(* PLC project Generated.project, CODESYS CODESYS V3.5 SP19 Patch 1 *)
(* stored: creationDateTime 2026-09-14T14:47:22.341572, modificationDateTime 2026-09-14T14:47:22.341572 *)

(* ═══════════════════════════════════════════════════════════════ ⚙️ ST_CycleMachineHomingCfg — Réglages IHM du cycle de référencement machine ─────────────────────────────────────────────────────────────── 🎯 Mise en service. Les réglages géométriques (positions capteur, offsets benne) restent portés par GVL_PERSISTENT (_WinchM1CfgPersist / _BucketCfgPersist). 💾 Ponté vers persist (_CycleMachineHomingCfgPersist) via FB_CfgPersistBridge_CycleMachineHomingCfg. ═══════════════════════════════════════════════════════════════ *)
TYPE ST_CycleMachineHomingCfg : STRUCT
  ForceStepTarget : INT := 0;  (* 🔧 Step GRAFCET cible du forçage (0=HX0 .. 9=HXF), borné côté FB *)
  Initialized : BOOL := FALSE;  (* 🚦 flag restauration boot *)
END_STRUCT;
END_TYPE

(* ======================================================================= 💾 FB_CfgPersistBridge_CycleMachineHomingCfg — Pont persistance pour ST_CycleMachineHomingCfg ─────────────────────────────────────────────────────────────── 🎯 Rôle : Restauration et synchronisation bidirectionnelle IHM / Persist 💾 Persistance : Transfert GVL_PERSISTENT <-> GVL_IHM sur Initialized 📄 Doc métier : DOC/AF/AF_Partie-03_Contrats_Composants_v2.3.md §3 ======================================================================= *)
FUNCTION_BLOCK FB_CfgPersistBridge_CycleMachineHomingCfg
  VAR_OUTPUT
    JustRestored : BOOL;  (* === ETATS RESTAURATION === <-- [STAT] Vrai sur le cycle de restauration initiale *)
  END_VAR
  VAR_IN_OUT
    Hmi : ST_CycleMachineHomingCfg;  (* === BUS CONFIGURATION ET PERSISTANCE === <-> [BUS] Structure de configuration IHM *)
    Persist : ST_CycleMachineHomingCfg;  (* <-> [BUS] Structure de configuration persistante *)
  END_VAR

            

JustRestored := FALSE;
IF NOT Hmi.Initialized THEN
    Hmi := Persist;
    Hmi.Initialized := TRUE;
    JustRestored := TRUE;
ELSE
    Persist := Hmi;
END_IF;

          
END_FUNCTION_BLOCK
